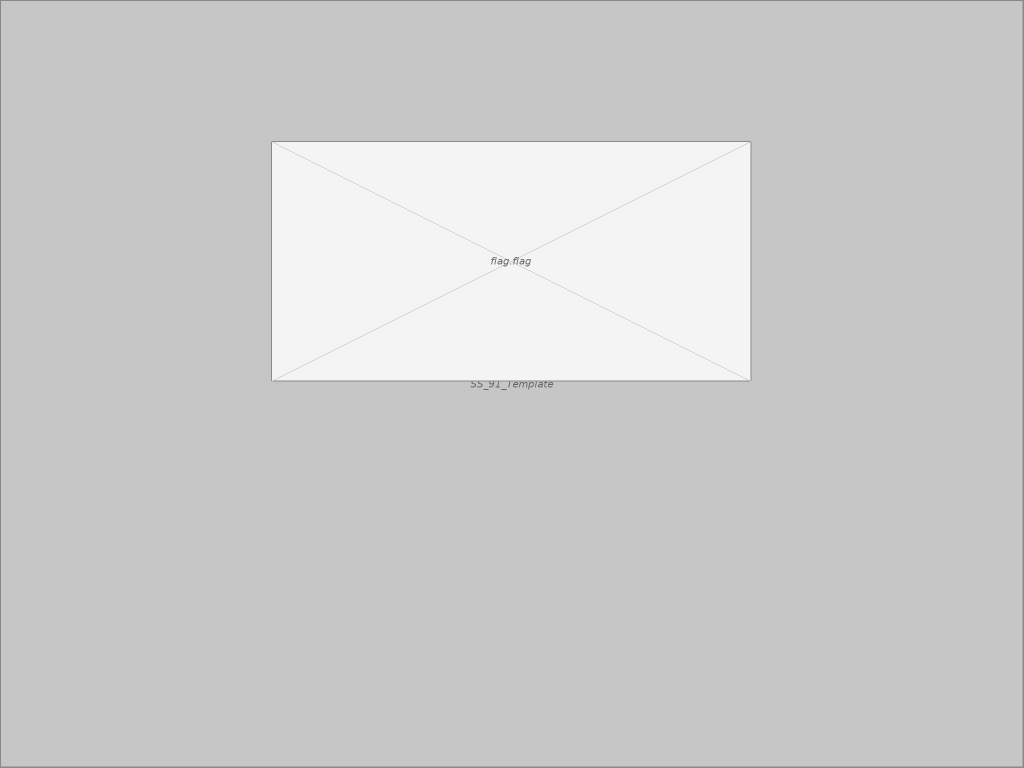
VISUALIZATION Mc_90_About  // 1024x768
    Frame (0,0 1024x768)
        shows SS_91_Template(header := gHMIData.hmiHeader)
    Image (271,141 480x240), image: flag.flag
END_VISUALIZATION

(* stored: Version 1.1.0.1, ProductVersion 3.1.4024.12
   Visu Mc_90_About: Id {8ef145eb-bbe7-43e6-a3a5-394ba62db052} *)
